{attribute 'qualified_only'}
VAR_GLOBAL
	Axis1 : AXIS_REF;
	
END_VAR

(* stored: Version 1.1.0.1, ProductVersion 3.1.4024.4
   GVL Global_Servo: Id {25a4cf3b-9e62-46ea-8af5-9f8bc37e5cf9} *)
